// Load stacker HW inputs
TYPE ST_InputsMovableStop :
STRUCT	
	HW				: ST_HW_InputsMovableStop;	// Hardware inputs
	CtrlIn			: ST_CtrlInMovableStop;		// ser function control inputs	
END_STRUCT
END_TYPE

(* stored: Version 1.1.0.1, ProductVersion 3.1.4024.9
   DUT ST_InputsMovableStop: Id {018ab452-6f5a-40fc-9de1-1ee1c46d8443} *)
